// TIA Portal V19 export
TYPE "C501_STU_NME_TYPIC"
   STRUCT
      OBS { ExternalAccessible := 'False'; ExternalVisible := 'False'; ExternalWritable := 'False'} : USInt;   // Niveaumeting in of uit dienst zetten
   END_STRUCT;
END_TYPE
